// TwinCAT 3 PLC project Untitled1
// ProgramVersion: 3.1.4026.17
// libraries:
//   Tc2_Standard, * (Beckhoff Automation GmbH)
//   Tc2_System, * (Beckhoff Automation GmbH)
//   Tc3_DriveMotionControl, * (Beckhoff Automation GmbH)
// project tree:
//   / PlcTask.TcTTO
//   POUs/ MAIN.TcPOU
// real-time tasks:
//   TASK PlcTask: cycle T#10ms, priority 20, ADS port 350
// I/O:
//   DEVICE Device 1 (EtherCAT), AmsNetId 5.146.234.225.2.1
//     Term 1 (EK1200) [EK1200-5000 EtherCAT Power supply (2A E-Bus)]
//       Term 2 (EL7062) [EL7062-0000 2Ch. Stepper motor output stage (48V, 3A)]
//         startup 32785:27 := 6C030000 // DRV Motor Settings Ch.1 / Motor speed limitation
//         startup 28688:3 := 08 // DRV Outputs Ch.1 / Modes of operation
//         startup 28688:16 := FF7F // DRV Outputs Ch.1 / Positive torque limit value
//         startup 28688:17 := FF7F // DRV Outputs Ch.1 / Negative torque limit value
//         startup 32784:87 := 64 // DRV Amplifier Settings Ch.1 / Position loop velocity feed forward gain
//         startup 32784:109 := 64000000 // DRV Amplifier Settings Ch.1 / Torque feed forward gain
//         startup 32785:52 := 70170000 // DRV Motor Settings Ch.1 / Configured motor current
//         startup 32784:19 := 1D00 // DRV Amplifier Settings Ch.1 / Current loop proportional gain
//         startup 32784:18 := 1E00 // DRV Amplifier Settings Ch.1 / Current loop integral time
//         startup 32784:21 := 91000000 // DRV Amplifier Settings Ch.1 / Velocity loop proportional gain
//         startup 32784:20 := 96000000 // DRV Amplifier Settings Ch.1 / Velocity loop integral time
//         startup 32776:18 := 0100 // FB Settings ENC Ch.1 / Encoder type
//         startup 32784:100 := 12 // DRV Amplifier Settings Ch.1 / Commutation type
//       Term 3 (EL1008) [EL1008 8Ch. Dig. Input 24V, 3ms]
//       Term 4 (EL2008) [EL2008 8Ch. Dig. Output 24V, 0.5A]
//       Term 5 (EL9011) [EL9011 End Terminal]
// variable links:
//   Untitled1/Untitled1 Instance <-> Device 1 (EtherCAT)/Term 1 (EK1200)/Term 2 (EL7062)
//     PlcTask Inputs/MAIN.Axis1.DriveToPlc <-> DMC Inputs Channel 1/DMC
//     PlcTask Inputs/MAIN.Axis1.InfoData/AdsAddr <-> InfoData/AdsAddr
//     PlcTask Inputs/MAIN.Axis1.InfoData/State <-> InfoData/State
//     PlcTask Inputs/MAIN.Axis1.WcState/InputToggle <-> WcState/InputToggle
//     PlcTask Inputs/MAIN.Axis1.WcState/WcState <-> WcState/WcState
//     PlcTask Outputs/MAIN.Axis1.PlcToDrive <-> DMC Outputs Channel 1/DMC
//   Untitled1/Untitled1 Instance <-> Device 1 (EtherCAT)/Term 1 (EK1200)/Term 3 (EL1008)
//     PlcTask Inputs/MAIN.bInput <-> Channel 1/Input

CONFIGURATION Untitled1
    RESOURCE PLC ON TwinCAT3
        TASK PlcTask(INTERVAL := T#10ms, PRIORITY := 20);
        PROGRAM MAIN WITH PlcTask : MAIN;
    END_RESOURCE
END_CONFIGURATION

// ---- POUs/MAIN.TcPOU
PROGRAM MAIN
VAR
	bInput AT%I*:BOOL;
	Axis1:AXIS_REF;
	MC_Power: MC_Power;
	bEnable: BOOL;
	MC_MoveAbsolute: MC_MoveAbsolute;
	bMove: BOOL;
END_VAR

Axis1.ReadStatus();

Axis1.Parameter.EncoderScalingFactor := 0.000000083819031715393066;;

Axis1.Parameter.MaxVelocity	:= 6000;

MC_Power(
	Axis:=Axis1 , 
	Enable:=bEnable , 
	Status=> , 
	Busy=> , 
	Active=> , 
	Error=> , 
	ErrorID=> );

MC_MoveAbsolute(
	Axis:=Axis1 , 
	Execute:=bMove , 
	Position:=0.0 , 
	Velocity:=100 , 
	Acceleration:=100 , 
	Deceleration:=100 , 
	Options:= , 
	Done=> , 
	Busy=> , 
	Active=> , 
	CommandAborted=> , 
	Error=> , 
	ErrorID=> );

END_PROGRAM
